FUNCTION_BLOCK PICKER_HMI (* Composite Function Block Type *)
  (* Standard: 61499-2 *)
  (* Version 0.2, 2003-12-05, JHC, Rockwell Automation, Renamed from NEWCOMPFB. *)
  (* Version 0.1, 2002-01-08, JHC, Rockwell Automation, Added DLY FB as example. *)
  (* Version 0.0, 2000-05-27, JHC, Rockwell Automation *)
  (* Compiler header: package fb.rt.pnp;import fb.rt.hmi.*; *)
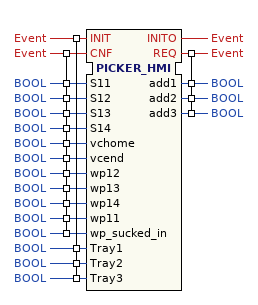
  EVENT_INPUT
    INIT WITH Tray1, Tray2, Tray3;
    CNF WITH S11, S12, S13, S14, vchome, vcend, wp12, wp13, wp14, wp11, wp_sucked_in; (* Confirmation from Plug *)
  END_EVENT
  EVENT_OUTPUT
    INITO;
    REQ WITH add1, add2, add3; (* Request from Socket *)
  END_EVENT
  VAR_INPUT
    S11 : BOOL;
    S12 : BOOL;
    S13 : BOOL;
    S14 : BOOL;
    vchome : BOOL;
    vcend : BOOL;
    wp12 : BOOL;
    wp13 : BOOL;
    wp14 : BOOL;
    wp11 : BOOL;
    wp_sucked_in : BOOL;
    Tray1 : BOOL;
    Tray2 : BOOL;
    Tray3 : BOOL;
  END_VAR
  VAR_OUTPUT
    add1 : BOOL;
    add2 : BOOL;
    add3 : BOOL;
  END_VAR
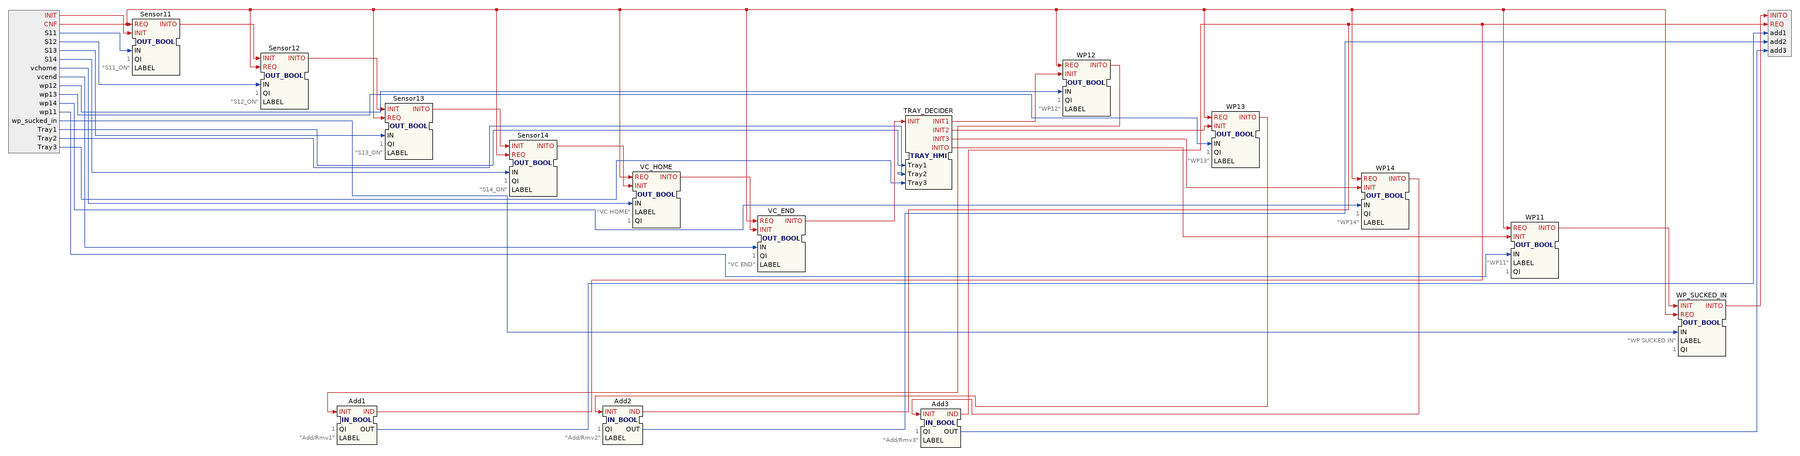
  FBS
    WP14 : OUT_BOOL(QI := 1, LABEL := "WP14");
    WP11 : OUT_BOOL(LABEL := "WP11", QI := 1);
    WP_SUCKED_IN : OUT_BOOL(LABEL := "WP SUCKED IN", QI := 1);
    VC_HOME : OUT_BOOL(LABEL := "VC HOME", QI := 1);
    VC_END : OUT_BOOL(QI := 1, LABEL := "VC END");
    WP12 : OUT_BOOL(QI := 1, LABEL := "WP12");
    WP13 : OUT_BOOL(QI := 1, LABEL := "WP13");
    Sensor11 : OUT_BOOL(QI := 1, LABEL := "S11_ON");
    Sensor12 : OUT_BOOL(QI := 1, LABEL := "S12_ON");
    Sensor13 : OUT_BOOL(QI := 1, LABEL := "S13_ON");
    Sensor14 : OUT_BOOL(QI := 1, LABEL := "S14_ON");
    Add1 : IN_BOOL(QI := 1, LABEL := "Add/Rmv1");
    Add2 : IN_BOOL(QI := 1, LABEL := "Add/Rmv2");
    Add3 : IN_BOOL(QI := 1, LABEL := "Add/Rmv3");
    TRAY_DECIDER : TRAY_HMI;
  END_FBS
  EVENT_CONNECTIONS
    CNF TO WP14.REQ;
    WP11.INITO TO WP_SUCKED_IN.INIT;
    CNF TO WP11.REQ;
    CNF TO WP_SUCKED_IN.REQ;
    CNF TO VC_HOME.REQ;
    CNF TO VC_END.REQ;
    CNF TO WP12.REQ;
    CNF TO WP13.REQ;
    Sensor11.INITO TO Sensor12.INIT;
    Sensor12.INITO TO Sensor13.INIT;
    Sensor13.INITO TO Sensor14.INIT;
    CNF TO Sensor11.REQ;
    CNF TO Sensor12.REQ;
    CNF TO Sensor13.REQ;
    CNF TO Sensor14.REQ;
    INIT TO Sensor11.INIT;
    Sensor14.INITO TO VC_HOME.INIT;
    VC_HOME.INITO TO VC_END.INIT;
    Add1.IND TO REQ;
    Add2.IND TO REQ;
    Add3.IND TO REQ;
    VC_END.INITO TO TRAY_DECIDER.INIT;
    TRAY_DECIDER.INIT1 TO WP12.INIT;
    TRAY_DECIDER.INIT2 TO WP13.INIT;
    TRAY_DECIDER.INIT3 TO WP14.INIT;
    TRAY_DECIDER.INITO TO WP11.INIT;
    WP12.INITO TO Add1.INIT;
    WP13.INITO TO Add2.INIT;
    WP14.INITO TO Add3.INIT;
    WP_SUCKED_IN.INITO TO INITO;
  END_CONNECTIONS
  DATA_CONNECTIONS
    S11 TO Sensor11.IN;
    S12 TO Sensor12.IN;
    S13 TO Sensor13.IN;
    S14 TO Sensor14.IN;
    vchome TO VC_HOME.IN;
    vcend TO VC_END.IN;
    wp12 TO WP12.IN;
    wp13 TO WP13.IN;
    wp14 TO WP14.IN;
    wp11 TO WP11.IN;
    wp_sucked_in TO WP_SUCKED_IN.IN;
    Add1.OUT TO add1;
    Add2.OUT TO add2;
    Add3.OUT TO add3;
    Tray1 TO TRAY_DECIDER.Tray1;
    Tray2 TO TRAY_DECIDER.Tray2;
    Tray3 TO TRAY_DECIDER.Tray3;
  END_CONNECTIONS
END_FUNCTION_BLOCK
